(* IEC 61131-3 sources: Std_PalletMover/Class/PeripheralBasicLift, 1 file *)

(* ---- PeripheralBasicLift.st ---- *)
(*!
<Class
	Name               = "PeripheralBasicLift"
	Revision           = "0.0"
	RealtimeTask       = "false"
	CyclicTask         = "false"
	BackgroundTask     = "false"
	Sigmatek           = "false"
	OSInterface        = "false"
	HighPriority       = "false"
	Automatic          = "false"
	UpdateMode         = "Prescan"
	SharedCommandTable = "true"
	Objectsize         = "(870,120)">
	<Channels>
		<Server Name="ActualHeight" Visualized="false" Initialize="false" WriteProtected="true" Retentive="false"/>
		<Server Name="Ain_ActualHeight" Visualized="false" Initialize="false" WriteProtected="true" Retentive="false"/>
		<Server Name="Bin_MaxHeight" Visualized="false" Initialize="false" WriteProtected="true" Retentive="false"/>
		<Server Name="Bin_MinHeight" Visualized="false" Initialize="false" WriteProtected="true" Retentive="false"/>
		<Server Name="ClassSvr" Visualized="false" Initialize="false" WriteProtected="true" Retentive="false"/>
		<Server Name="SetHeight" Visualized="false" Initialize="false" WriteProtected="true" Retentive="false"/>
		<Server Name="SetSpeed" Visualized="false" Initialize="false" WriteProtected="true" Retentive="false"/>
		<Server Name="State" Visualized="false" Initialize="false" WriteProtected="true" Retentive="false"/>
		<Server Name="ToObject" Class="PeripheralsBase" Visualized="false" Initialize="false" WriteProtected="true" Retentive="false" Comment="ToObject:&#13;&#10;Object channel server.&#13;&#10;Channel to reach the methodes of this object.&#13;&#10;&#13;&#10;In case this object should be Accessible by a pointer&#13;&#10;the variable ToObject is used to handover the address of this object.&#13;&#10;&#13;&#10;This server is never used for anything else!!!&#13;&#10;&#13;&#10;&#13;&#10;"/>
		<Client Name="AgvConfig" Required="true" Internal="false"/>
		<Client Name="AgvSettings" Required="true" Internal="false"/>
		<Client Name="I_Lift" Required="true" Internal="true"/>
		<Client Name="ObjPeripheral" Required="true" Internal="true"/>
		<Client Name="op_LogData" Required="false" Internal="false" Comment="Output for logging data to SF_Logger"/>
		<Client Name="p_NextObject" Required="false" Internal="false" Comment="Pointer to next object in linked list"/>
	</Channels>
	<Separators>
		<Servers>
			<SepChn Position="6"/>
		</Servers>
	</Separators>
	<Network Name="PeripheralBasicLift">
		<!-- List of Components in this network -->
		<Components>
			<Object
				Name       = "I_Lift"
				Class      = "I_Lift"
				Position   = "(870,180)"
				Visualized = "false">
				<Channels>
					<Server Name="ActualHeight"/>
					<Server Name="ClassSvr"/>
					<Server Name="SetHeight"/>
					<Server Name="SetSpeed"/>
					<Server Name="State"/>
				</Channels>
			</Object>
			<Object
				Name       = "ObjPeripheral"
				Class      = "PeripheralsBase"
				Position   = "(120,180)"
				Visualized = "false">
				<Channels>
					<Server Name="ToObject"/>
					<Client Name="op_LogData"/>
					<Client Name="p_NextObject"/>
				</Channels>
			</Object>
		</Components>
		<Comments>
		</Comments>
		<!-- List of Connections in this network -->
		<Connections>
			<Connection Source="this.ObjPeripheral" Destination="ObjPeripheral.ToObject"/>
			<Connection Source="this.I_Lift" Destination="I_Lift.ClassSvr"/>
			<Connection Source="this.ActualHeight" Destination="I_Lift.ActualHeight" Vertices="(1958,330),(1786,330),"/>
			<Connection Source="this.SetHeight" Destination="I_Lift.SetHeight" Vertices="(1958,390),(1786,390),"/>
			<Connection Source="this.SetSpeed" Destination="I_Lift.SetSpeed" Vertices="(1958,450),(1786,450),"/>
			<Connection Source="this.State" Destination="I_Lift.State" Vertices="(1958,510),(1786,510),"/>
			<Connection Source="ObjPeripheral.p_NextObject" Destination="this.p_NextObject" Vertices="(120,330),(38,330),"/>
			<Connection Source="ObjPeripheral.op_LogData" Destination="this.op_LogData" Vertices="(120,270),(30,420),(38,390),"/>
			<Connection Source="this.ToObject" Destination="ObjPeripheral.ToObject" Vertices="(1958,270),(706,270),"/>
		</Connections>
		<!-- Headerfiles -->
		<Options>
		</Options>
	</Network>
</Class>
*)
PeripheralBasicLift : CLASS
  //Servers:
	ClassSvr 	: SvrChCmd_DINT;
	ToObject 	: SvrChCmd_pVoid;
	ActualHeight 	: SvrCh_DINT;
	SetHeight 	: SvrCh_DINT;
	SetSpeed 	: SvrCh_DINT;
	State 	: SvrCh_LiftState_PTofCls_I_Lift;
	Ain_ActualHeight 	: SvrCh_DINT;
	Bin_MaxHeight 	: SvrCh_DINT;
	Bin_MinHeight 	: SvrCh_DINT;
  //Clients:
	ObjPeripheral 	: CltChCmd_PeripheralsBase;
	I_Lift 	: CltChCmd_I_Lift;
	AgvConfig 	: CltChCmd_AgvConfig;
	AgvSettings 	: CltChCmd_AgvSettings;
	p_NextObject 	: CltChCmd_LinkedObjectBase;
	op_LogData 	: CltCh_gpt_LogData;
  //Variables:
  //Functions:

	FUNCTION VIRTUAL GLOBAL ToObject::Read
		VAR_OUTPUT
			output (EAX) 	: pVoid;
		END_VAR;

	FUNCTION VIRTUAL GLOBAL ActualHeight::Read
		VAR_OUTPUT
			output (EAX) 	: DINT;
		END_VAR;

	FUNCTION VIRTUAL GLOBAL SetHeight::Read
		VAR_OUTPUT
			output (EAX) 	: DINT;
		END_VAR;

	FUNCTION VIRTUAL GLOBAL SetSpeed::Read
		VAR_OUTPUT
			output (EAX) 	: DINT;
		END_VAR;

	FUNCTION VIRTUAL GLOBAL State::Read
		VAR_OUTPUT
			output (EAX) 	: I_Lift::LiftState;
		END_VAR;
  //Tables:
	FUNCTION @STD
		VAR_OUTPUT
			ret_code	: CONFSTATES;
		END_VAR;
	FUNCTION GLOBAL TAB @CT_;
END_CLASS;

#pragma using I_Lift
#pragma using PeripheralsBase
#pragma usingLtd AgvConfig
#pragma usingLtd AgvSettings
#pragma usingLtd LinkedObjectBase

FUNCTION VIRTUAL GLOBAL PeripheralBasicLift::ActualHeight::Read
	VAR_OUTPUT
		output (EAX) 	: DINT;
	END_VAR

	ActualHeight := I_Lift.ActualHeight.Read();
	output := ActualHeight;

END_FUNCTION

FUNCTION VIRTUAL GLOBAL PeripheralBasicLift::SetHeight::Read
	VAR_OUTPUT
		output (EAX) 	: DINT;
	END_VAR

	SetHeight := I_Lift.SetHeight.Read();
	output := SetHeight;

END_FUNCTION

FUNCTION VIRTUAL GLOBAL PeripheralBasicLift::SetSpeed::Read
	VAR_OUTPUT
		output (EAX) 	: DINT;
	END_VAR

	SetSpeed := I_Lift.SetSpeed.Read();
	output := SetSpeed;

END_FUNCTION

FUNCTION VIRTUAL GLOBAL PeripheralBasicLift::State::Read
	VAR_OUTPUT
		output (EAX) 	: I_Lift::LiftState;
	END_VAR

	State := I_Lift.State.Read();
	output := State;

END_FUNCTION

FUNCTION VIRTUAL GLOBAL PeripheralBasicLift::ToObject::Read
	VAR_OUTPUT
		output (EAX) 	: pVoid;
	END_VAR

	ToObject := ObjPeripheral.ToObject.Read();
	output := ToObject;

END_FUNCTION
